// TIA Portal V20 export
TYPE "LER_typeStatusEm1"
// stored: Access Published
   STRUCT
      dancerValueChanged : Bool;
      dancerMode : Int := 2;
      dancerHighKp : LReal := 2.0;
      dancerHighIntegTime : LReal := 0.0;
      dancerHighLimit : LReal := 10.0;
      dancerLowKp : LReal := 0.8;
      dancerLowIntegTime : LReal := 0.0;
      dancerLowLimit : LReal := 5.0;
   END_STRUCT;
END_TYPE
